KUKA KRL program: SET_DEFAULT_IMPED.src

&ACCESS RVO2
&REL 18
&PARAM TEMPLATE = C:\KRC\Roboter\Template\FunctionVorgabe
&PARAM EDITMASK = *
DEFFCT BOOL SET_DEFAULT_IMPED( )

DECL STIFFNESS USERSTIFF
USERSTIFF = $STIFFNESS
USERSTIFF.FRAMETYPE=#BASE
USERSTIFF.STRATEGY = 20
USERSTIFF.CPSTIFFNESS = {X 2000.0, Y 2000.0, Z 2000.0, A 200.0, B 200.0, C 200.0}
USERSTIFF.CPDAMPING = {X 0.7, Y 0.7, Z 0.7, A 0.7, B 0.7, C 0.7}
USERSTIFF.AXISSTIFFNESS = {A1 1000.0, A2 1000.0, A3 1000.0, A4 1000.0, A5 1000.0, A6 1000.0, E1 1000.0}
USERSTIFF.AXISDAMPING = {A1 0.7, A2 0.7, A3 0.7, A4 0.7, A5 0.7, A6 0.7, E1 0.7}
USERSTIFF.CPMAXDELTA = {X 100.0, Y 100.0, Z 100.0, A 20.0, B 20.0, C 20.0}
USERSTIFF.MAXFORCE = {X 70.0, Y 70.0, Z 70.0, A 10.0, B 10.0, C 10.0}
USERSTIFF.AXISMAXDELTA = {A1 10.0, A2 10.0, A3 10.0, A4 10.0, A5 10.0, A6 10.0, E1 10.0}
USERSTIFF.AXISMAXDELTATRQ = {A1 2.0, A2 2.0, A3 2.0, A4 2.0, A5 2.0, A6 2.0, E1 2.0}

$STIFFNESS = USERSTIFF

RETURN TRUE

ENDFCT
